FUNCTION_BLOCK FB_OH_SensorControl
VAR_INPUT
	FunctionNumber	: E_FunctionNumber;
	ZoneNumber		: INT;
	OH_PositionSide	: INT; //1,2,3 or 4
	OH_SensorInput	: BOOL;
	Mute			: BOOL; //mutes test when it is not needed, e.g. when group is not active
END_VAR
VAR_OUTPUT
END_VAR
VAR_IN_OUT
	Error		: ST_ErrorDataSet;  
END_VAR
VAR
	TransportData	: ST_TransportControlData;
	OH_SensorOK		: BOOL;
	TakeoverActive	: BOOL;
	HandoverActive	: BOOL;   
	CheckOverhang	: BOOL;
	CheckToggle		: BOOL; 
	Fwd				: BOOL; 
END_VAR

TransportData := F_PB_GetTransportControlDataRef(FunctionNumber,ZoneNumber);
CheckOverhang := TRUE;
CheckToggle	  := FALSE;

//Function data valid
IF NOT( FunctionNumber > E_FunctionNumber.F_BEGIN_FUNCTION AND FunctionNumber < E_FunctionNumber.F_END_FUNCTION) THEN
	F_SetError(
		ErrorType	:= E_ErrorType.ERROR,
		ErrorParam	:= 'Function number not defined',
		ErrorMsg 	:= E_ErrorConv.CONFIGURATION_ERROR,
		ErrorData	:= Error);
END_IF

//Zone number valid 
IF( ZoneNumber < 1 OR ZoneNumber > NUMBER_OF_ZONES_PER_FUNCTION) THEN
		F_SetError(
			ErrorType	:= E_ErrorType.ERROR,
			ErrorParam	:= 'Zone number not defined',
			ErrorMsg 	:= E_ErrorConv.CONFIGURATION_ERROR,
			ErrorData	:= Error);
END_IF

//Uses OR in order to stay active even if the transport is interrupted
TakeoverActive := TakeoverActive OR TransportData.eTakeOverState = E_TakeOverState.ACTIVE;
HandoverActive := HandoverActive OR TransportData.eHandOverState = E_HandOverState.ACTIVE;

//Decide direction, True Forward, False reverse
Fwd := F_IsFwdDriveDirection(FunctionNumber, TakeoverActive, HandoverActive); 

IF TakeoverActive THEN 
	IF( Fwd AND (OH_PositionSide = 1 OR OH_PositionSide = 3)) OR 
		(NOT Fwd AND (OH_PositionSide = 2 OR OH_PositionSide = 4)) THEN
		
		CheckOverhang := FALSE;
		CheckToggle	  := TRUE;
		IF NOT OH_SensorInput THEN
			//If OH sensor was toggled
			OH_SensorOK := TRUE;
		END_IF
	END_IF
END_IF

IF HandoverActive THEN
	IF( Fwd AND (OH_PositionSide = 2 OR OH_PositionSide = 4)) OR 
		(NOT Fwd AND (OH_PositionSide = 1 OR OH_PositionSide = 3)) THEN
		
		CheckOverhang := FALSE;
		CheckToggle	  := TRUE;
		IF NOT OH_SensorInput THEN
			//If OH sensor was toggled
			OH_SensorOK := TRUE;
		END_IF
	END_IF
END_IF

//When takeover or handover is complete
IF( TransportData.Occupied AND TakeoverActive) OR
	(NOT TransportData.Occupied AND HandoverActive) THEN 

	IF NOT OH_SensorOK AND CheckToggle THEN 
		F_SetError(
				ErrorType	:= E_ErrorType.ERROR,
				ErrorParam	:= CONCAT('OH sensor not broken side: ', TO_STRING(OH_PositionSide)),
				ErrorMsg 	:= E_ErrorConv.INCORRECT_SENSOR_SIGNAL,
				ErrorData	:= Error);
	END_IF
	
	//Test completed, reset values
	TakeoverActive := FALSE;
	HandoverActive := FALSE;
	OH_SensorOK := FALSE;

END_IF

//Check IF sensor is blocked
IF CheckOverhang AND NOT Mute THEN 
	IF( NOT OH_SensorInput) THEN 
	//Overhang sensors blocked
	F_SetError(
			ErrorType	:= E_ErrorType.ERROR,
			ErrorParam	:= CONCAT(CONCAT('OH sensor side: ', TO_STRING(OH_PositionSide)),' blocked'),
			ErrorMsg 	:= E_ErrorConv.INCORRECT_SENSOR_SIGNAL,
			ErrorData	:= Error);
	END_IF
END_IF

END_FUNCTION_BLOCK

(* stored: Version 1.1.0.1, ProductVersion 3.1.4024.9
   POU FB_OH_SensorControl: Id {c82365a7-24e7-4fc1-bca5-fcf7117b44c3}, SpecialFunc None *)
